{attribute addProperty BoxType "EPP2316-0003-0016"}
{attribute addProperty Id "OutputAT %Q*ARRAY[0 ..7] OF BOOL6480"}
{attribute addProperty CRC "1062725746"}
{attribute addProperty SizeInBites "64"}
{attribute addProperty SizeInBytes "8"}
TYPE DIG_Outputs_33B76376 :
STRUCT
	{attribute addProperty Name "Output"}
	Output AT %Q* : ARRAY[0 ..7] OF BOOL;
END_STRUCT
END_TYPE

(* stored: Version 1.2.0.0, ProductVersion 3.1.4024.9
   DUT DIG_Outputs_33B76376: Id {0dbc871e-32b2-4e50-8d26-a3200f119f33} *)
